Fanuc KAREL source: kt00503.KL

-- PROVISIONAL review KL for V940-1; original PC SHA256 8d50aee12c7fe1dce0e47581cd870df4cfb5d9d54c6515a36720047044fdaa17
-- Incomplete behavior may be omitted. Consult companion uncertainty JSON. Do not deploy.
PROGRAM KT00503
%NOLOCKGROUP
VAR
  OUT : BOOLEAN
-- UNRESOLVED_DECL P1 type=000102
-- UNRESOLVED_DECL P2 type=000106
BEGIN
  -- V9_ZERO_TABLE_METADATA_HINT layout=0001; no indexed target words; source/name/runtime held
  -- UNRESOLVED_PC offsets 5-20; opcodes 2E,22,32,35
  -- UNRESOLVED_PC offsets 25-40; opcodes 2E,22,32,35
  -- UNRESOLVED_PC offsets 45-78; opcodes 49,7E,49,7E,AC,23
  -- UNRESOLVED_PC offsets 83-87; opcodes 7F
END KT00503
